FUNCTION_BLOCK FB_TurnTableService EXTENDS FB_ActionBasic
VAR_INPUT
    xExecute      : BOOL;
    xAbort        : BOOL;
    iTurnTableTarget : INT;			//1=A ,2=B ,3=C ,4=D
    Cylinder : REFERENCE TO UNI_CylinderList;
    TimeOut  : LREAL := 30; // Unit : s
END_VAR
VAR_OUTPUT
    xAborted : BOOL;
    iErrorID : INT;
    ErrorMsg : STRING;
END_VAR
VAR
    StateBehavior   : CBML.ETrigATo;
    CurrentPosition : ST_PositionTable;
	uiCyclicStep    : UINT := 0;
	PosCmd			: INT;
END_VAR

THIS^.IBehaviourModel := StateBehavior;
StateBehavior(xExecute := xExecute,
              xAbort := xAbort,
              udiTimeOut := LREAL_TO_UDINT( TimeOut*1000000),
              xDone => xDone,
              xBusy => xBusy,
              xError => xError,
              xAborted => xAborted);
			  
//Error Msg
iErrorID := StateBehavior._model.iErrorID;
ErrorMsg := M_GetErrorMsg(xErrorID := iErrorID);

METHOD CleanupAction
VAR_INPUT
    xAbortProposed : BOOL;
    iErrorIDProposed: INT;
END_VAR
VAR_OUTPUT
    xComplete : BOOL := TRUE;
    xAbort: BOOL := xAbortProposed;
 	iErrorID : INT := iErrorIDProposed;
END_VAR
END_METHOD

METHOD CyclicAction
VAR_INPUT
    itfTimingController : CBML.ITimingController;
END_VAR
VAR_OUTPUT
    xComplete : BOOL := TRUE;
    iErrorID : INT := 0;
END_VAR
VAR_INST
	
END_VAR
xComplete := FALSE;
CASE uiCyclicStep OF
    0:
		Cylinder.List.fbTurntable_Press.M_Retract();

        IF Cylinder.List.fbTurntable_Press.InRearPosition THEN
            uiCyclicStep := 100;
        END_IF
    100:
        arAxisCtrl_gb[AxisNo.TurnTable].PosMode.Position := PosCmd;
		

        IF arAxisStatus_gb[AxisNo.TurnTable].Admin._OpModeAck = ModePosAbs AND arAxisStatus_gb[AxisNo.TurnTable].Admin.CmdDone THEN
            uiCyclicStep := 200;
        END_IF
	200:
        Cylinder.List.fbTurntable_Press.M_Extend();

        IF Cylinder.List.fbTurntable_Press.InFrontPosition THEN
            xComplete := TRUE;
        END_IF
END_CASE

IF arAxisCtrl_gb[AxisNo.TurnTable].Admin.Axis.Status.Error THEN
    iErrorID := 6; // Axis TurnTable has error
END_IF

//IF Cylinder.List.fbTurntable_Press.xError THEN
//    iErrorID := 7;	//Clinder Error
//END_IF
END_METHOD

METHOD ExitAction
VAR_INPUT
    xAfterCleanup : BOOL;
    xInCopyCode : BOOL;
END_VAR
END_METHOD

METHOD M_GetErrorMsg : T_MaxString
VAR_INPUT
	xErrorID: INT;
END_VAR

VAR
	
END_VAR
CASE xErrorID OF
	0:
		M_GetErrorMsg := 'No Error';
	1:
		M_GetErrorMsg := 'Action time out';
	2:
		M_GetErrorMsg := 'Position Data invalid';
	3:
		M_GetErrorMsg := 'TurnTableTarget invalid';
	4:
		M_GetErrorMsg := 'Axis not ready';
	5:
		M_GetErrorMsg := 'Cylinder not ready';
	6:
		M_GetErrorMsg := 'Axis TurnTable has Error';
	7:
		M_GetErrorMsg := 'fbTurntable_Press has Error';
END_CASE
END_METHOD

METHOD ResetAction
VAR_OUTPUT
    xComplete : BOOL := TRUE;
END_VAR
END_METHOD

METHOD StartAction
VAR_OUTPUT
    xComplete : BOOL := TRUE;
	iErrorID : INT := 0;
END_VAR
xComplete := FALSE;
IF NOT (iTurnTableTarget >= 1 AND iTurnTableTarget <= 4) THEN
    iErrorID := 3; // Target Station invalid.
    RETURN;
END_IF

IF NOT arAxisCtrl_gb[AxisNo.TurnTable].Admin.Axis.Status.NotMoving AND
     arAxisCtrl_gb[AxisNo.TurnTable].Admin.Axis.Status.Error THEN
    iErrorID := 4; // Axis not ready
END_IF

CASE iTurnTableTarget OF 
	1:	//A
		PosCmd :=0;
		xComplete := TRUE;
	2:	//B
		PosCmd :=270;
		xComplete := TRUE;
	3:	//C
		PosCmd :=180;
		xComplete := TRUE;
	4:	//D
		PosCmd :=90;
		xComplete := TRUE;
END_CASE


//IF Cylinder.List.fbTurntable_Press.xBusy AND  
//NOT Cylinder.List.fbTurntable_Press.xError  THEN
//	iErrorID := 5; // Cylinder not ready
//END_IF

uiCyclicStep := 0;
END_METHOD

END_FUNCTION_BLOCK

(* stored: Version 1.1.0.1, ProductVersion 3.1.4024.13
   POU FB_TurnTableService: Id {4bd385a0-9f51-4e07-9759-c8ce4665575d}, SpecialFunc None
   Folder Action: Id {a5765f18-10fd-4fc9-b3a9-88b0bdffd540}
   Method CleanupAction: Id {ce35767d-b1db-45dc-aa8f-da5d40e8e7bb}
   Method CyclicAction: Id {cc1f20f7-e0b1-460a-9e13-0e2b3f8dfa6d}
   Method ExitAction: Id {5a085846-80be-40c5-90c9-c1d06e06b59f}
   Method M_GetErrorMsg: Id {716a5a99-61df-4633-9b52-c4c5677c75a7}
   Method ResetAction: Id {9e96d1c2-4ebe-4a38-9037-fe33ecf144af}
   Method StartAction: Id {fc86e512-b248-440c-bfcc-c96402127e9c} *)
